PROGRAM P_Linked_List
VAR
END_VAR

P_Singly_Linked_List();
P_Doubly_Linked_List();

END_PROGRAM

(* stored: Version 1.1.0.1, ProductVersion 3.1.4024.4
   POU P_Linked_List: Id {f61c3acb-991b-491b-b0a4-6beac0b2bf6d}, SpecialFunc None *)
